FUNCTION_BLOCK E_T_FF (* Toggle flip flop *)
  (* Standard: 61499-1 Annex A; Description: Copyright (c) 2017 fortiss GmbH This program and the accompanying materials are made available under the terms of the Eclipse Public License 2.0 which is available at https://www.eclipse.org/legal/epl-2.0/ SPDX-License-Identifier: EPL-2.0 *)
  (* Version 1.0, 2017-09-22, Alois Zoitl, fortiss GmbH, initial API and implementation and/or initial documentation *)
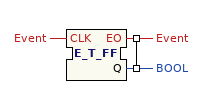
  EVENT_INPUT
    CLK; (* Clock for triggering a output toggle *)
  END_EVENT
  EVENT_OUTPUT
    EO WITH Q; (* Output Q has changed *)
  END_EVENT
  VAR_OUTPUT
    Q : BOOL; (* value of flip flop *)
  END_VAR
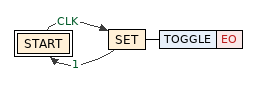
  EC_STATES
    START; (* Initial State *)
    SET : TOGGLE -> EO; (* Initialization *)
  END_STATES
  EC_TRANSITIONS
    START TO SET := CLK;
    SET TO START := 1;
  END_TRANSITIONS
  ALGORITHM TOGGLE IN ST: (* TOGGLE algorithm *)
Q := NOT Q;
  END_ALGORITHM
END_FUNCTION_BLOCK
